{region '#Template'}
	{attribute 'Version' := '6.0.0.0'}
	{attribute 'Tags' := '"LCID": "1031", "Text": "RA, Sunprotection, Sunblind"'}
	{attribute 'Tags' := '"LCID": "1033", "Text": "RA, Sunprotection, Sunblind"'}
	{attribute 'Using' := '"Type": "Template", "URI": "BA2_Param"'}
	{attribute 'Using' := '"Type": "Template", "URI": "ST_BA_SunblindActuatorFeedback"'}
	{attribute 'Description' := '"LCID": "1031", "Text": "Sonnenschutzaktor (Jalousie)"'}
	{attribute 'Description' := '"LCID": "1033", "Text": "Sunblind-actuator (venetian blind)"'}
{endregion}
FUNCTION_BLOCK FB_BA_SunBld EXTENDS FB_BA_View


VAR_INPUT
	bEn						: BOOL;
	stSunBldCmd				: ST_BA_SunBld;		// Low-Priorities command telegram
END_VAR
VAR_OUTPUT
	bReferencing			: BOOL;				// device is being referenced
	nReferenceTimer			: UDINT;            
	bErr					: BOOL;				// error
	fActualPosition			: REAL;				// actual position
	fActualAngle			: REAL;				// actual angle
	eActualSunblindPrio		: BYTE;				// actual telegram priority
	stFeedback				: ST_BA_SunblindActuatorFeedback;
END_VAR
VAR_INPUT CONSTANT PERSISTENT
	{attribute 'parameterUnit':= 'ms'}
	nSwiOverTi 				: UDINT;
	{attribute 'parameterUnit':= 'ms'}
	nPositioningDelay		: UDINT;	// delay of automatic telegrams [ms] to prevent overload
	{attribute 'parameterUnit':= 'ms'}  
	nTiUp					: UDINT;	// total driving-up-time [ms]
	{attribute 'parameterUnit':= 'ms'}  
	nTiDwn					: UDINT;	// total driving-down-time [ms]
	{attribute 'parameterUnit':= 'ms'}          		
	nTurnTiUp				: UDINT;	// time to turn lamellas up [ms]
	{attribute 'parameterUnit':= 'ms'}          		
	nTurnTiDwn				: UDINT;	// time to turn lamellas down [ms]
	{attribute 'parameterUnit':= 'ms'}          		
	nBckLshTiUp				: UDINT;	// Time to traverse the backlash in the upward direction [ms]
	{attribute 'parameterUnit':= 'ms'}          		
	nBckLshTiDwn			: UDINT;	// Time to traverse the backlash in the downward direction [ms]
	{attribute 'parameterUnit':= 'deg'} 
	fAnglLmtUp				: REAL;		// upper limit of lamellas in deg - must be greater than fAnglLmtDwn
	{attribute 'parameterUnit':= 'deg'} 
	fAnglLmtDwn				: REAL;		// lower limit of lamellas in deg - must be lower than fAnglLmtUp
END_VAR
VAR_INPUT CONSTANT				 
	ActualPosition			: FB_BA_AV_Op;		
	ActualAngle				: FB_BA_AV_Op;		
END_VAR
VAR
	PositioningDelay		: FB_BA_SunBldPosDly;
	SunBldActr				: FB_BA_SunBldActr;
	bCmdUp			AT %Q*	: BOOL;
	bCmdDown		AT %Q*	: BOOL;
END_VAR
VAR // added by the converter: edge detectors and wires of the graphical bodies
    _s1 : ST_BA_SunblindActuatorFeedback;
END_VAR

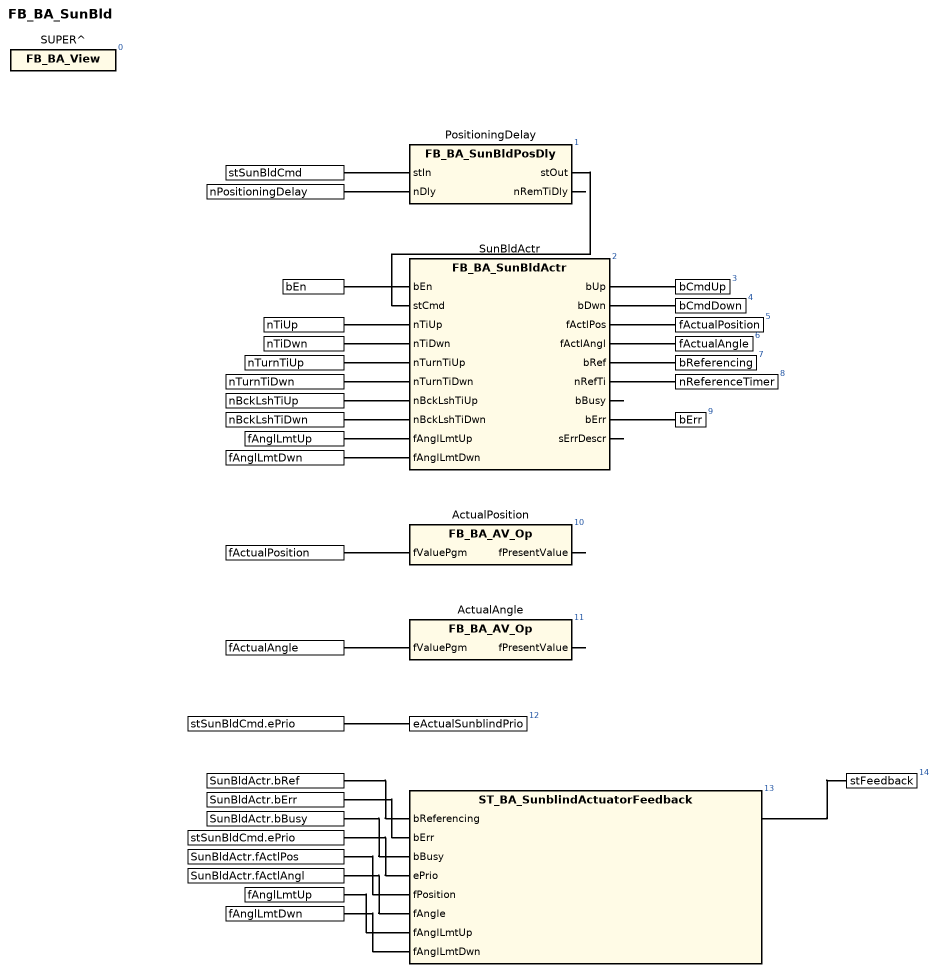
SUPER^(); // FB_BA_View
PositioningDelay(stIn := stSunBldCmd, nDly := nPositioningDelay); // FB_BA_SunBldPosDly
SunBldActr(
    bEn := bEn,
    stCmd := PositioningDelay.stOut,
    nTiUp := nTiUp,
    nTiDwn := nTiDwn,
    nTurnTiUp := nTurnTiUp,
    nTurnTiDwn := nTurnTiDwn,
    nBckLshTiUp := nBckLshTiUp,
    nBckLshTiDwn := nBckLshTiDwn,
    fAnglLmtUp := fAnglLmtUp,
    fAnglLmtDwn := fAnglLmtDwn); // FB_BA_SunBldActr
bCmdUp := SunBldActr.bUp;
bCmdDown := SunBldActr.bDwn;
fActualPosition := SunBldActr.fActlPos;
fActualAngle := SunBldActr.fActlAngl;
bReferencing := SunBldActr.bRef;
nReferenceTimer := SunBldActr.nRefTi;
bErr := SunBldActr.bErr;
ActualPosition(fValuePgm := fActualPosition); // FB_BA_AV_Op
ActualAngle(fValuePgm := fActualAngle); // FB_BA_AV_Op
eActualSunblindPrio := stSunBldCmd.ePrio;
// compose _s1 : ST_BA_SunblindActuatorFeedback
_s1.bReferencing := SunBldActr.bRef;
_s1.bErr := SunBldActr.bErr;
_s1.bBusy := SunBldActr.bBusy;
_s1.ePrio := stSunBldCmd.ePrio;
_s1.fPosition := SunBldActr.fActlPos;
_s1.fAngle := SunBldActr.fActlAngl;
_s1.fAnglLmtUp := fAnglLmtUp;
_s1.fAnglLmtDwn := fAnglLmtDwn;
stFeedback := _s1;

METHOD FB_init : BOOL
VAR_INPUT
	bInitRetains : BOOL; // if TRUE; the retain variables are initialized (warm start / cold start)
	bInCopyCode : BOOL;  // if TRUE; the instance afterwards gets moved into the copy code (online change)
END_VAR
nSwiOverTi 						:= 250;			// switch-over-time of manual actuator
nPositioningDelay				:= 250;			// delay of automatic telegrams [ms] to prevent overload
nTiUp							:= 50000;		// total driving-up-time [ms]
nTiDwn							:= 50000;		// total driving-down-time [ms]
nTurnTiUp						:= 1500;		// time to turn lamellas up [ms]
nTurnTiDwn						:= 1500;		// time to turn lamellas down [ms]
nBckLshTiUp						:= 100;			// Time to traverse the backlash in the upward direction [ms]
nBckLshTiDwn					:= 100;			// Time to traverse the backlash in the downward direction [ms]
fAnglLmtUp						:= 30;			// upper limit of lamellas in deg - must be greater than fAnglLmtDwn
fAnglLmtDwn						:= -70;			// lower limit of lamellas in deg - must be lower than fAnglLmtUp

// actual position / aktueller Position
ActualPosition.iParent			:= THIS^;
ActualPosition.iLabel			:= LblFun_FeedbackSunblindPosition;
ActualPosition.eUnit			:= E_BA_Unit.eOther_Percent;
ActualPosition.fCOVIncrement	:= BA2_Param.fDefCOVIncrement;

// actual angle / aktueller Lamellenwinkel
ActualAngle.iParent				:= THIS^;
ActualAngle.iLabel				:= LblFun_FeedbackSunblindAngle;
ActualAngle.eUnit				:= E_BA_Unit.eOther_DegreesAngular;
ActualAngle.fCOVIncrement		:= BA2_Param.fDefCOVIncrement;
END_METHOD

END_FUNCTION_BLOCK

(* stored: Version 1.1.0.1, ProductVersion 3.1.4024.12
   POU FB_BA_SunBld: Id {90427cbb-0820-42bb-b619-398b532b3312}, SpecialFunc None
   Method FB_init: Id {8990c953-7053-40b2-b879-ce23d3025bbd} *)
